Fanuc KAREL source: PAUSE_TASK.kl

PROGRAM T
%NOLOCKGROUP
VAR
 v0 : STRING[40]
 v1 : BOOLEAN
 v2 : BOOLEAN
 v3 : INTEGER
BEGIN
 PAUSE_TASK(v0, v1, v2, v3)
END T
